{attribute addProperty BoxType "AX8206-0000-0041-0041"}
{attribute addProperty Id "Ch_B_Target_positionAT %Q*DINT3240Ch_B_Target_velocityAT %Q*DINT3240"}
{attribute addProperty CRC "3927654880"}
{attribute addProperty SizeInBites "64"}
{attribute addProperty SizeInBytes "8"}
TYPE Ch_B_Interpolator_Outputs_EA1B41E0 :
STRUCT
	{attribute addProperty Name "Ch_B_Target_position"}
	Ch_B_Target_position AT %Q* : DINT;
	{attribute addProperty Name "Ch_B_Target_velocity"}
	Ch_B_Target_velocity AT %Q* : DINT;
END_STRUCT
END_TYPE

(* stored: Version 1.2.0.0, ProductVersion 3.1.4024.9
   DUT Ch_B_Interpolator_Outputs_EA1B41E0: Id {031de8f5-4cac-48f6-8c36-83944d7ca52e} *)
